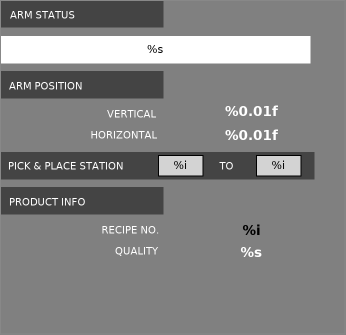
VISUALIZATION Popup_ArmInfo  // 346x335
    Rectangle (0,0 346x335)
    RoundedRectangle (0,36 310x27), "%s", text variable: sStatusMessage
    Rectangle (0,0 163x27)
    Label (7,3 152x24), "ARM STATUS"
    Rectangle (0,152 314x27)
    Label (5,158 172x16), "PICK & PLACE STATION"
    Rectangle (158,155 45x21), "%i", text variable: ARDSGnrFeedArmPnpParameter[1].iPickStationNo
    Label (204,154 45x24), "TO"
    Rectangle (256,155 45x21), "%i", text variable: ARDSGnrFeedArmPnpParameter[1].iTransferStationNo
    Rectangle (0,71 163x27)
    Label (6,74 152x24), "ARM POSITION"
    Label (9,102 150x24), "VERTICAL"
    Label (9,123 151x24), "HORIZONTAL"
    Rectangle (0,187 163x27)
    Label (6,190 153x24), "PRODUCT INFO"
    Label (11,218 151x24), "RECIPE NO."
    Label (13,239 148x24), "QUALITY"
    Rectangle (167,103 169x17), "%0.01f", text variable: DSArm1VertConfig.lrGen_Out_CurrentPos
    Rectangle (167,127 169x17), "%0.01f", text variable: DSArm1HorzConfig.lrGen_Out_CurrentPos
    Rectangle (167,222 169x17), "%i", text variable: DSArmBasketInfo[1].iProductRecipeNo
        OnMouseDown: write the text variable via VisuDialogs.Numpad
    Rectangle (167,244 169x17), "%s", text variable: DSArmBasketInfo[1].sProductQuality
END_VISUALIZATION

(* stored: Version 1.1.0.1, ProductVersion 3.1.4024.12
   Visu Popup_ArmInfo: Id {268f1fb7-ebe0-49f3-a7f9-35e2c44b6a77} *)
